{attribute 'qualified_only'}
{attribute 'strict'}
TYPE E_RobotArmJointDirection :
(
	LEFT	:= 1,
	RIGHT	:= 2
);
END_TYPE

(* stored: Version 1.1.0.1, ProductVersion 3.1.4024.9
   DUT E_RobotArmJointDirection: Id {0de8fc1a-c2f5-4caf-abc5-42bd4f3783ea} *)
